KUKA KRL program: palletizing.src, palletizing.dat

--- palletizing.src ---
&ACCESS RVO
DEF  palletizing ( )

DECL INT row, col, maxRow, maxCol
DECL REAL dX, dY, dZ
DECL E6POS placePosition, upPosition

;FOLD INI;%{PE}
  ;FOLD BASISTECH INI
    GLOBAL INTERRUPT DECL 3 WHEN $STOPMESS==TRUE DO IR_STOPM ( )
    INTERRUPT ON 3
    BAS (#INITMOV,0 )
  ;ENDFOLD (BASISTECH INI)
  ;FOLD USER INI
    ;Make your modifications here

  ;ENDFOLD (USER INI)
;ENDFOLD (INI)

;FOLD PTP HOME  Vel= 100 % DEFAULT;%{PE}%MKUKATPBASIS,%CMOVE,%VPTP,%P 1:PTP, 2:HOME, 3:, 5:100, 7:DEFAULT
$BWDSTART = FALSE
PDAT_ACT=PDEFAULT
FDAT_ACT=FHOME
BAS (#PTP_PARAMS,100 )
$H_POS=XHOME
PTP  XHOME
;ENDFOLD

maxRow = 3
maxCol = 3
dX = 58
dY = 39
dZ = 120

FOR row = 1 to maxRow
   for col = 1 to maxCol
      pickstone()

      placePosition = XP1
      placePosition.X = placePosition.X + (row-1)*dX
      placePosition.Y = placePosition.Y + (col-1)*dY

      upPosition = placePosition
      upPosition.Z = upPosition.Z + dZ

      $TOOL = TOOL_DATA[14]
      $BASE = BASE_DATA[5]

      SPTP upPosition
      SLIN placePosition

      GRPg_SetStateAndCheck(1,1,0.2,0)

      SLIN upPosition

   endfor
endfor

FOR row = maxRow to 1 STEP -1


   for col = maxCol to 1 STEP -1

      GRPg_SetStateAndCheck(1,1,0.2,0)

      placePosition = XP1
      placePosition.X = placePosition.X + (row-1)*dX
      placePosition.Y = placePosition.Y + (col-1)*dY

      upPosition = placePosition
      upPosition.Z = upPosition.Z + dZ

      $TOOL = TOOL_DATA[14]
      $BASE = BASE_DATA[5]

      SPTP upPosition
      SLIN placePosition

      GRPg_SetStateAndCheck(1, 2, 0.2, 1)

      SLIN upPosition

      storestone()

   endfor
endfor

;FOLD PTP HOME  Vel= 100 % DEFAULT;%{PE}%MKUKATPBASIS,%CMOVE,%VPTP,%P 1:PTP, 2:HOME, 3:, 5:100, 7:DEFAULT
$BWDSTART = FALSE
PDAT_ACT=PDEFAULT
FDAT_ACT=FHOME
BAS (#PTP_PARAMS,100 )
$H_POS=XHOME
PTP  XHOME
;ENDFOLD

END

--- palletizing.dat ---
&ACCESS RVO
DEFDAT  palletizing
;FOLD EXTERNAL DECLARATIONS;%{PE}%MKUKATPBASIS,%CEXT,%VCOMMON,%P
;FOLD BASISTECH EXT;%{PE}%MKUKATPBASIS,%CEXT,%VEXT,%P
EXT  BAS (BAS_COMMAND  :IN,REAL  :IN )
DECL INT SUCCESS
;ENDFOLD (BASISTECH EXT)
;FOLD USER EXT;%{E}%MKUKATPUSER,%CEXT,%VEXT,%P
;Make your modifications here

;ENDFOLD (USER EXT)
;ENDFOLD (EXTERNAL DECLARATIONS)
DECL E6POS XP1={X 53.5255089,Y 31.8043327,Z -37.8078613,A -121.298653,B 88.1064072,C -32.0049706,S 2,T 10,E1 0.0,E2 0.0,E3 0.0,E4 0.0,E5 0.0,E6 0.0}
DECL FDAT FP1={TOOL_NO 14,BASE_NO 5,IPO_FRAME #BASE,POINT2[] " ",TQ_STATE FALSE}
ENDDAT
